FUNCTION CurrentToRaw : UINT

VAR_INPUT
  amps : REAL;           // 0.00 to 5.00
END_VAR

VAR
  tmp : REAL; // 0 to 5000
END_VAR


tmp := amps * 1000.0;

IF tmp < 0.0 THEN
	tmp := 0.0;
ELSIF tmp > 5000.0 THEN
	tmp := 5000.0;
END_IF;

CurrentToRaw := REAL_TO_UINT(tmp);

END_FUNCTION

(* stored: Version 1.1.0.1
   POU CurrentToRaw: Id {08ef05f9-463e-4bda-b3a7-c03a9456ce66}, SpecialFunc None *)
